// TIA Portal V17 export
// export: Created 2023-12-22T15:03:02.9337006Z, ExportSetting WithDefaults, DisplayName Totally Integrated Automation Portal, DisplayVersion V17, DisplayName TIA Portal Openness, DisplayVersion V17, DisplayName TIA Portal Version Control Interface, DisplayVersion V17, DisplayName STEP 7 Professional, DisplayVersion V17, DisplayName STEP 7 Safety, DisplayVersion V17, DisplayName WinCC Advanced, DisplayVersion V17
DATA_BLOCK "AO_example_DB"   // DB400
VERSION : 0.1
// stored: AutoNumber false, DBAccessibleFromOPCUA true, DBAccessibleFromWebserver true, InstanceOfName AO_ex, InstanceOfType FB
"AO_ex"
   // VAR_INPUT
   //    SP_A : Real;
   //    All_Block : Bool;
   // END_VAR
   // VAR_IN_OUT
   //    Signal : Int;
   // END_VAR
   // VAR RETAIN
   //    CMD : "CMD";
   //    Mode : Int;
   //    Status : Int;
   //    Use : Struct
   //       Indirect { S7_SetPoint := 'True'} : Bool := TRUE;
   //    END_STRUCT;
   //    VmA : Real;
   //    SP_M : Real;
   //    Converter { S7_SetPoint := 'True'} : "Converter_LAD";
   //    Events : Word;
   //    pos : Array[0..15] of Bool;
   //    Output_Type { S7_SetPoint := 'True'} : Int := 0;
   //    CodeID { S7_SetPoint := 'True'} : Int := 0;
   //    "Type" { S7_SetPoint := 'True'} : Int := 0;
   //    ADDR { S7_SetPoint := 'True'} : Int := 0;
   //    Slow { S7_SetPoint := 'True'} : "Slow";
   //    Time_DTL { S7_SetPoint := 'True'} : DTL := DTL#2023-05-02-18:36:48.766257666;
   // END_VAR
BEGIN
   Converter.Use_Min_In := FALSE;
   Converter.Use_Max_In := FALSE;
   Converter.Use_Min_Out := FALSE;
   Converter.Use_Max_Out := FALSE;
   Converter.IO := FALSE;
   Converter.Inverse := FALSE;
   Converter.Min_In := 0.0;
   Converter.Min_Out := 0.0;
   Converter.Max_In := 0.0;
   Converter.Max_Out := 0.0;
   Slow.Use_Up := FALSE;
   Slow.Use_Down := FALSE;
   Slow.Step_Up := 0.125;
   Slow.Step_Down := 0.125;
   Slow.T_Up.SP := 1.0;
   Slow.T_Up.One := 0.1;
   Slow.T_Down.SP := 1.0;
   Slow.T_Down.One := 0.1;
END_DATA_BLOCK
